TYPE ST_St020_HMI_OUT :
STRUCT
	//Trolley	: ST_Trolley;
END_STRUCT
END_TYPE

(* stored: Version 1.1.0.1
   DUT ST_St020_HMI_OUT: Id {299c9d92-bc26-44c5-a34e-a48352e8a395} *)
